// TIA Portal V18 export
DATA_BLOCK "HMI_DB"   // DB15
{ S7_Optimized_Access := 'TRUE' }
// stored: MemoryReserve 100
   VAR
      CS_Homing : Bool;
      CS_PP_Reset : Bool;
      CS_PL_Reset : Bool;
      CS_TP_Reset : Bool;
      CS_TL_Reset : Bool;
      CS_Virtual_Reset : Bool;
      CS_Reset : Bool;
      CS_PP_Power : Bool;
      CS_PL_Power : Bool;
      CS_TP_Power : Bool;
      CS_TL_Power : Bool;
      CS_Virtual_Power : Bool;
      CS_Power : Bool;
   END_VAR
BEGIN
END_DATA_BLOCK
